(* PLC project Unnamed, Unknown Unnamed 1 *)
(* stored: creationDateTime 2024-05-10T13:42:21, modificationDateTime 2024-05-10T14:22:13 *)

PROGRAM Logic_Gates
  VAR
    Input_0 : BOOL;
    Input_1 : BOOL;
    Input_2 : BOOL;
    Input_3 : BOOL;
    Input_4 : BOOL;
    Output_0 : BOOL;
    Output_1 : BOOL;
    Output_2 : BOOL;
  END_VAR

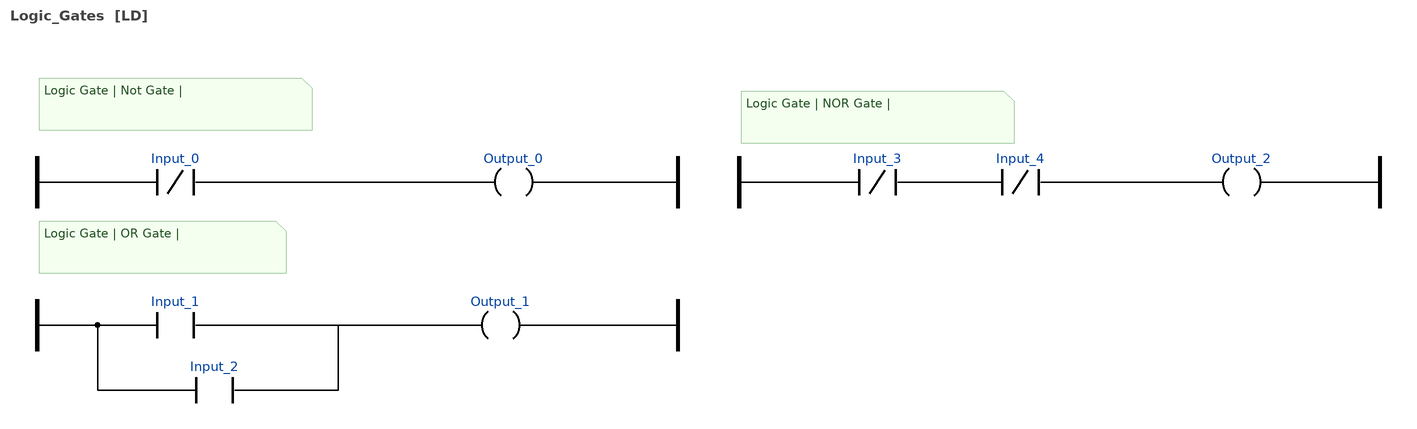
(* LD diagram, written out as Structured Text *)
(* Logic Gate | Not Gate | *)
(* Logic Gate | NOR Gate | *)
Output_0 := NOT Input_0;
(* Logic Gate | OR Gate | *)
Output_1 := Input_1 OR Input_2;
Output_2 := NOT Input_3 AND NOT Input_4;
END_PROGRAM

CONFIGURATION Config0
  RESOURCE Res0 ON PLC
    TASK task0(INTERVAL := T#20ms, PRIORITY := 0);
    PROGRAM instance0 WITH task0 : Logic_Gates;
  END_RESOURCE
END_CONFIGURATION
